// TIA Portal V16 export
// export: Created 2021-11-12T13:32:06.3227527Z, ExportSetting WithDefaults, DisplayName Totally Integrated Automation Portal, DisplayVersion V16 Update 3, DisplayName TIA Portal Version Control Interface, DisplayVersion V16 Update 2, DisplayName TIA Portal Openness, DisplayVersion V16 Update 3, DisplayName SINAMICS Startdrive Advanced, DisplayVersion V16 Update 5, DisplayName SINAMICS Startdrive G130, G150, S120, S150, SINAMICS MV, S210, DisplayVersion V16 Update 5, DisplayName SINAMICS Startdrive G110M, G120, G120C, G120D, G120P, G115D, DisplayVersion V16 Update 5, DisplayName STEP 7 Professional, DisplayVersion V16 Update 3, DisplayName STEP 7 Safety, DisplayVersion V16, DisplayName WinCC UA Professional, DisplayVersion V16 Update 3
FUNCTION_BLOCK "Station160"   // FB10, LAD
{ S7_Optimized_Access := 'TRUE' }
VERSION : 0.1
// stored: AutoNumber true, IsIECCheckEnabled false, IsRetainMemResEnabled false, MemoryReserve 100, SetENOAutomatically false, UDAEnableTagReadback false
   VAR
      STD_RobotZones : "STD_RobotZones";
      SI_PartType { S7_SetPoint := 'True'} : Int;
      SDI_PartID : DInt;
      SI_PartCounter : Int;
   END_VAR
   VAR_TEMP
      TI_RowNo : Int;
      TI_LineNo : Int;
      TB1IndexValid : Bool;
   END_VAR
   VAR CONSTANT
      CI_NrOfRows : Int := 24;
      CI_NrOfLines : Int := 2;
   END_VAR
   VAR_TEMP   // added for the SCL form of the ladder/FBD networks
      _w1 : Bool;
   END_VAR
BEGIN

REGION Network 1: ***************ClearTemporary***************
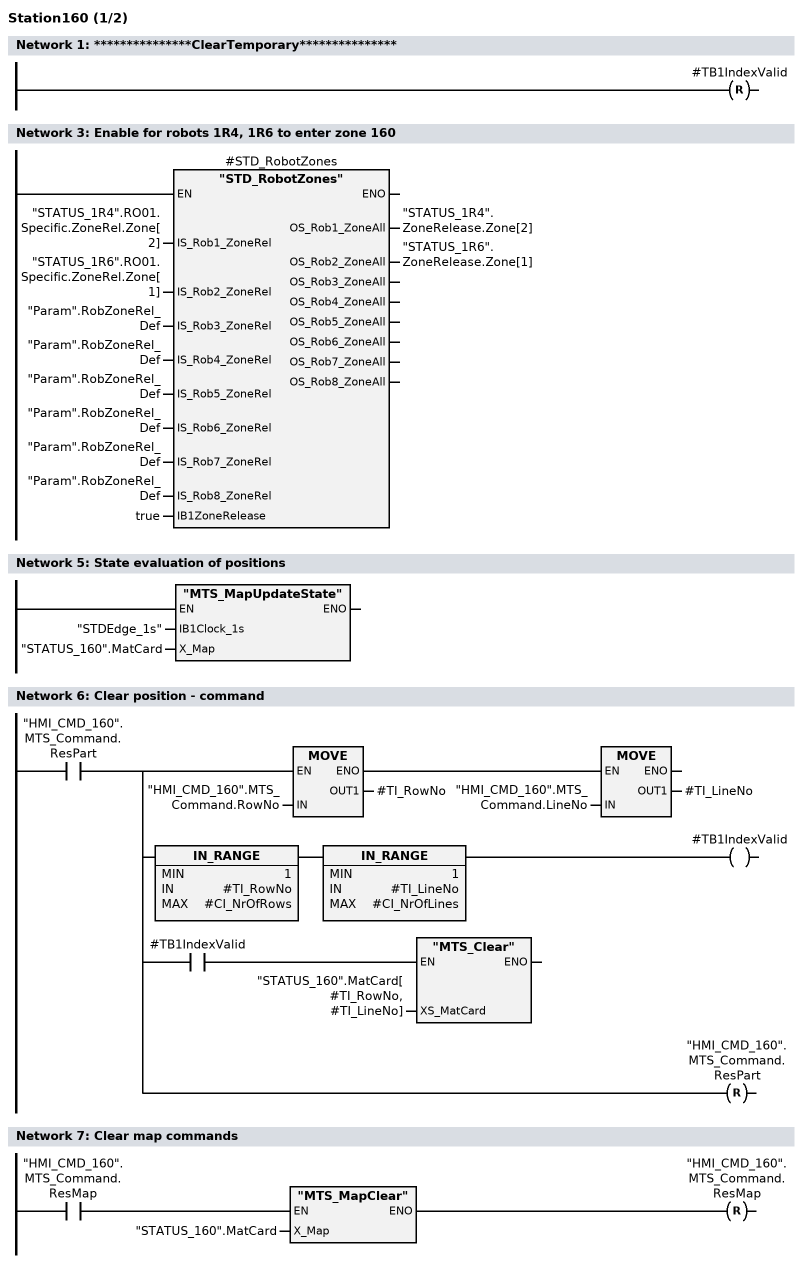
   RUNG wire#powerrail
      R_Coil( #TB1IndexValid )
   END_RUNG
   // the same network as SCL:
   #TB1IndexValid := FALSE;
END_REGION

REGION Network 2: *************** Robot zones ***************
END_REGION

REGION Network 3: Enable for robots 1R4, 1R6 to enter zone 160
   RUNG wire#powerrail
      #STD_RobotZones(IS_Rob1_ZoneRel := "STATUS_1R4".RO01.Specific.ZoneRel.Zone[2], IS_Rob2_ZoneRel := "STATUS_1R6".RO01.Specific.ZoneRel.Zone[1], IS_Rob3_ZoneRel := "Param".RobZoneRel_Def, IS_Rob4_ZoneRel := "Param".RobZoneRel_Def, IS_Rob5_ZoneRel := "Param".RobZoneRel_Def, IS_Rob6_ZoneRel := "Param".RobZoneRel_Def, IS_Rob7_ZoneRel := "Param".RobZoneRel_Def, IS_Rob8_ZoneRel := "Param".RobZoneRel_Def, IB1ZoneRelease := true, OS_Rob1_ZoneAll => "STATUS_1R4".ZoneRelease.Zone[2], OS_Rob2_ZoneAll => "STATUS_1R6".ZoneRelease.Zone[1], OS_Rob3_ZoneAll =>, OS_Rob4_ZoneAll =>, OS_Rob5_ZoneAll =>, OS_Rob6_ZoneAll =>, OS_Rob7_ZoneAll =>, OS_Rob8_ZoneAll =>)
   END_RUNG
   // the same network as SCL:
   #STD_RobotZones(IS_Rob1_ZoneRel := "STATUS_1R4".RO01.Specific.ZoneRel.Zone[2],   // "STD_RobotZones"
                   IS_Rob2_ZoneRel := "STATUS_1R6".RO01.Specific.ZoneRel.Zone[1],
                   IS_Rob3_ZoneRel := "Param".RobZoneRel_Def,
                   IS_Rob4_ZoneRel := "Param".RobZoneRel_Def,
                   IS_Rob5_ZoneRel := "Param".RobZoneRel_Def,
                   IS_Rob6_ZoneRel := "Param".RobZoneRel_Def,
                   IS_Rob7_ZoneRel := "Param".RobZoneRel_Def,
                   IS_Rob8_ZoneRel := "Param".RobZoneRel_Def,
                   IB1ZoneRelease := true,
                   OS_Rob1_ZoneAll => "STATUS_1R4".ZoneRelease.Zone[2],
                   OS_Rob2_ZoneAll => "STATUS_1R6".ZoneRelease.Zone[1]);
END_REGION

REGION Network 4: *************** Material flow ***************
END_REGION

REGION Network 5: State evaluation of positions
   RUNG wire#powerrail
      "MTS_MapUpdateState"(IB1Clock_1s := "STDEdge_1s", X_Map := "STATUS_160".MatCard)
   END_RUNG
   // the same network as SCL:
   "MTS_MapUpdateState"(IB1Clock_1s := "STDEdge_1s", X_Map := "STATUS_160".MatCard);
END_REGION

REGION Network 6: Clear position - command
   RUNG wire#powerrail
      Contact( "HMI_CMD_160".MTS_Command.ResPart )
      wire#w1
      Move(in := "HMI_CMD_160".MTS_Command.RowNo, out1 => #TI_RowNo)
      Move(in := "HMI_CMD_160".MTS_Command.LineNo, out1 => #TI_LineNo)
   END_RUNG
   RUNG wire#w1
      { S7_Templates := "SrcType := Int" } InRange(min := 1, in := #TI_RowNo, max := #CI_NrOfRows)
      { S7_Templates := "SrcType := Int" } InRange(min := 1, in := #TI_LineNo, max := #CI_NrOfLines)
      Coil( #TB1IndexValid )
   END_RUNG
   RUNG wire#w1
      Contact( #TB1IndexValid )
      "MTS_Clear"(XS_MatCard := "STATUS_160".MatCard[#TI_RowNo, #TI_LineNo])
   END_RUNG
   RUNG wire#w1
      R_Coil( "HMI_CMD_160".MTS_Command.ResPart )
   END_RUNG
   // the same network as SCL:
   IF "HMI_CMD_160".MTS_Command.ResPart THEN
       #TI_RowNo := "HMI_CMD_160".MTS_Command.RowNo;
       #TI_LineNo := "HMI_CMD_160".MTS_Command.LineNo;
   END_IF;
   #TB1IndexValid := "HMI_CMD_160".MTS_Command.ResPart AND (1 <= #TI_RowNo) AND (#TI_RowNo <= #CI_NrOfRows) AND (1 <= #TI_LineNo) AND (#TI_LineNo <= #CI_NrOfLines);
   #_w1 := "HMI_CMD_160".MTS_Command.ResPart;
   IF "HMI_CMD_160".MTS_Command.ResPart AND #TB1IndexValid THEN
       "MTS_Clear"(XS_MatCard := "STATUS_160".MatCard[#TI_RowNo, #TI_LineNo]);
   END_IF;
   IF #_w1 THEN "HMI_CMD_160".MTS_Command.ResPart := FALSE; END_IF;
END_REGION

REGION Network 7: Clear map commands
   RUNG wire#powerrail
      Contact( "HMI_CMD_160".MTS_Command.ResMap )
      "MTS_MapClear"(X_Map := "STATUS_160".MatCard)
      R_Coil( "HMI_CMD_160".MTS_Command.ResMap )
   END_RUNG
   // the same network as SCL:
   "MTS_MapClear"(EN := "HMI_CMD_160".MTS_Command.ResMap, X_Map := "STATUS_160".MatCard, ENO => #_w1);
   IF #_w1 THEN "HMI_CMD_160".MTS_Command.ResMap := FALSE; END_IF;
END_REGION

REGION Network 8: Set positions - init
   // "JSA0Comm" - change when recipes done
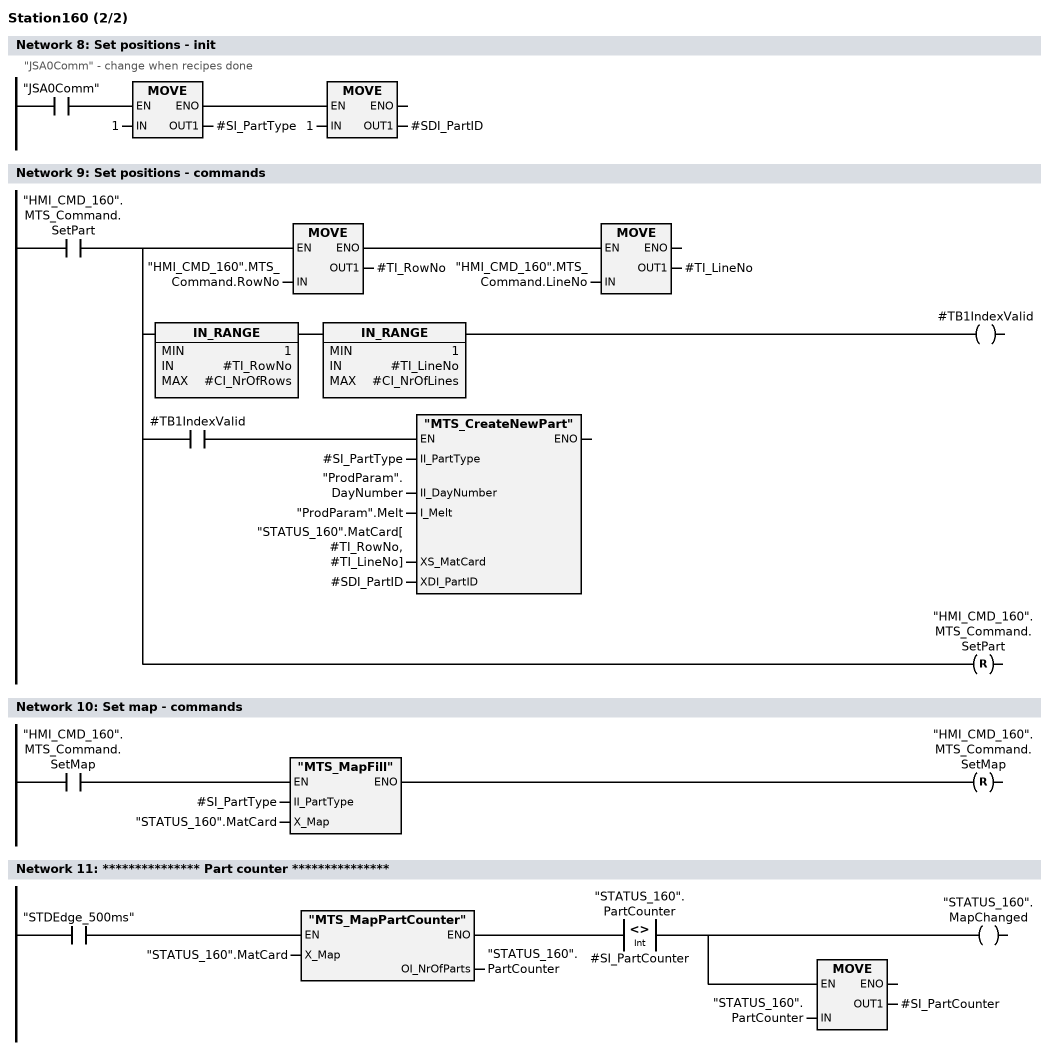
   RUNG wire#powerrail
      Contact( "JSA0Comm" )
      Move(in := 1, out1 => #SI_PartType)
      Move(in := 1, out1 => #SDI_PartID)
   END_RUNG
   // the same network as SCL:
   IF "JSA0Comm" THEN
       #SI_PartType := 1;
       #SDI_PartID := 1;
   END_IF;
END_REGION

REGION Network 9: Set positions - commands
   RUNG wire#powerrail
      Contact( "HMI_CMD_160".MTS_Command.SetPart )
      wire#w1
      Move(in := "HMI_CMD_160".MTS_Command.RowNo, out1 => #TI_RowNo)
      Move(in := "HMI_CMD_160".MTS_Command.LineNo, out1 => #TI_LineNo)
   END_RUNG
   RUNG wire#w1
      { S7_Templates := "SrcType := Int" } InRange(min := 1, in := #TI_RowNo, max := #CI_NrOfRows)
      { S7_Templates := "SrcType := Int" } InRange(min := 1, in := #TI_LineNo, max := #CI_NrOfLines)
      Coil( #TB1IndexValid )
   END_RUNG
   RUNG wire#w1
      Contact( #TB1IndexValid )
      "MTS_CreateNewPart"(II_PartType := #SI_PartType, II_DayNumber := "ProdParam".DayNumber, I_Melt := "ProdParam".Melt, XS_MatCard := "STATUS_160".MatCard[#TI_RowNo, #TI_LineNo], XDI_PartID := #SDI_PartID)
   END_RUNG
   RUNG wire#w1
      R_Coil( "HMI_CMD_160".MTS_Command.SetPart )
   END_RUNG
   // the same network as SCL:
   IF "HMI_CMD_160".MTS_Command.SetPart THEN
       #TI_RowNo := "HMI_CMD_160".MTS_Command.RowNo;
       #TI_LineNo := "HMI_CMD_160".MTS_Command.LineNo;
   END_IF;
   #TB1IndexValid := "HMI_CMD_160".MTS_Command.SetPart AND (1 <= #TI_RowNo) AND (#TI_RowNo <= #CI_NrOfRows) AND (1 <= #TI_LineNo) AND (#TI_LineNo <= #CI_NrOfLines);
   #_w1 := "HMI_CMD_160".MTS_Command.SetPart;
   IF "HMI_CMD_160".MTS_Command.SetPart AND #TB1IndexValid THEN
       "MTS_CreateNewPart"(II_PartType := #SI_PartType,
                           II_DayNumber := "ProdParam".DayNumber,
                           I_Melt := "ProdParam".Melt,
                           XS_MatCard := "STATUS_160".MatCard[#TI_RowNo, #TI_LineNo],
                           XDI_PartID := #SDI_PartID);
   END_IF;
   IF #_w1 THEN "HMI_CMD_160".MTS_Command.SetPart := FALSE; END_IF;
END_REGION

REGION Network 10: Set map - commands
   RUNG wire#powerrail
      Contact( "HMI_CMD_160".MTS_Command.SetMap )
      "MTS_MapFill"(II_PartType := #SI_PartType, X_Map := "STATUS_160".MatCard)
      R_Coil( "HMI_CMD_160".MTS_Command.SetMap )
   END_RUNG
   // the same network as SCL:
   "MTS_MapFill"(EN := "HMI_CMD_160".MTS_Command.SetMap,
                 II_PartType := #SI_PartType,
                 X_Map := "STATUS_160".MatCard,
                 ENO => #_w1);
   IF #_w1 THEN "HMI_CMD_160".MTS_Command.SetMap := FALSE; END_IF;
END_REGION

REGION Network 11: *************** Part counter ***************
   RUNG wire#powerrail
      Contact( "STDEdge_500ms" )
      "MTS_MapPartCounter"(X_Map := "STATUS_160".MatCard, OI_NrOfParts => "STATUS_160".PartCounter)
      { S7_Templates := "SrcType := Int" } NE_Contact(in1 := "STATUS_160".PartCounter, in2 := #SI_PartCounter)
      wire#w1
      Coil( "STATUS_160".MapChanged )
   END_RUNG
   RUNG wire#w1
      Move(in := "STATUS_160".PartCounter, out1 => #SI_PartCounter)
   END_RUNG
   // the same network as SCL:
   "MTS_MapPartCounter"(EN := "STDEdge_500ms",
                        X_Map := "STATUS_160".MatCard,
                        OI_NrOfParts => "STATUS_160".PartCounter,
                        ENO => #_w1);
   "STATUS_160".MapChanged := #_w1 AND ("STATUS_160".PartCounter <> #SI_PartCounter);
   IF "STATUS_160".MapChanged THEN #SI_PartCounter := "STATUS_160".PartCounter; END_IF;
END_REGION
END_FUNCTION_BLOCK
